% RSLogix 500 project P6.RSS, saved by version 12.00.00.00 %
PROJECT "UNTITLED"    % processor: Bul.1763 MicroLogix 1100 Series B %

PROGRAM FILES
  LAD 2 "MAIN"  3 rungs
  LAD 3 "DIGITAL IO"  2 rungs
  LAD 4 "CONTROL"  10 rungs

DATA FILES
  O0 OUTPUT  4 elements
  I1 INPUT  6 elements
  S2 STATUS  66 elements
  B3 BINARY  1 elements
  T4 TIMER  1 elements
  C5 COUNTER  3 elements
  R6 CONTROL  1 elements
  N7 INTEGER  4 elements
  F8 FLOAT  1 elements

LADDER 2 "MAIN"
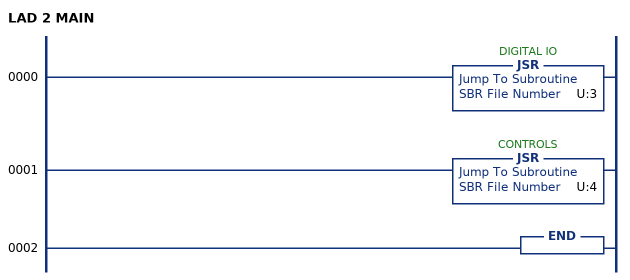
% Rung: 0 %
SOR JSR U:3 EOR
%   U:3  "DIGITAL IO" %
% Rung: 1 %
SOR JSR U:4 EOR
%   U:4  "CONTROLS" %
% Rung: 2 %
SOR END EOR

LADDER 3 "DIGITAL IO"
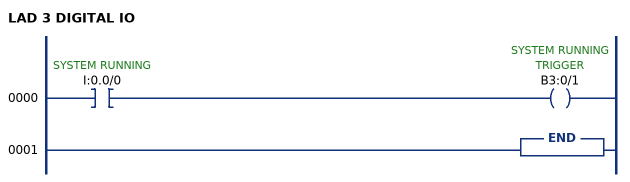
% Rung: 0 %
SOR XIC I:0.0/0 OTE B3:0/1 EOR
%   I:0.0/0  "SYSTEM RUNNING" %
%   B3:0/1  "SYSTEM RUNNING TRIGGER" %
% Rung: 1 %
SOR END EOR

LADDER 4 "CONTROL"
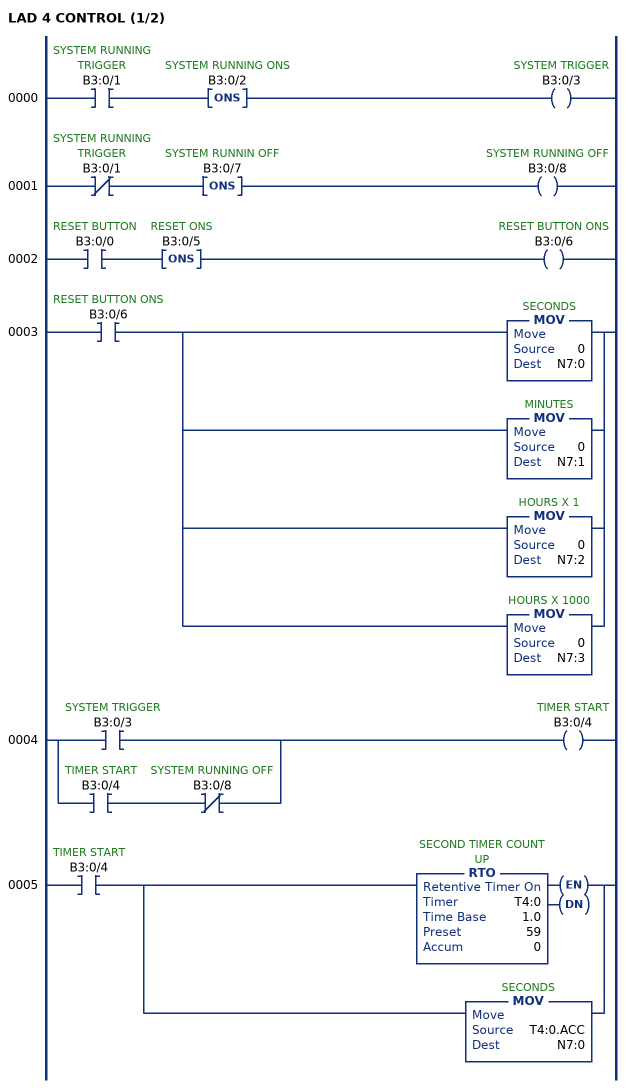
% Rung: 0 %
SOR XIC B3:0/1 ONS B3:0/2 OTE B3:0/3 EOR
%   B3:0/1  "SYSTEM RUNNING TRIGGER" %
%   B3:0/2  "SYSTEM RUNNING ONS" %
%   B3:0/3  "SYSTEM TRIGGER" %
% Rung: 1 %
SOR XIO B3:0/1 ONS B3:0/7 OTE B3:0/8 EOR
%   B3:0/1  "SYSTEM RUNNING TRIGGER" %
%   B3:0/7  "SYSTEM RUNNIN OFF" %
%   B3:0/8  "SYSTEM RUNNING OFF" %
% Rung: 2 %
SOR XIC B3:0/0 ONS B3:0/5 OTE B3:0/6 EOR
%   B3:0/0  "RESET BUTTON" %
%   B3:0/5  "RESET ONS" %
%   B3:0/6  "RESET BUTTON ONS" %
% Rung: 3 %
SOR XIC B3:0/6 BST MOV 0 N7:0 NXB MOV 0 N7:1 NXB MOV 0 N7:2 NXB MOV 0 N7:3 BND EOR
%   B3:0/6  "RESET BUTTON ONS" %
%   N7:0  "SECONDS" %
%   N7:1  "MINUTES" %
%   N7:2  "HOURS X 1" %
%   N7:3  "HOURS X 1000" %
% Rung: 4 %
SOR BST XIC B3:0/3 NXB XIC B3:0/4 XIO B3:0/8 BND OTE B3:0/4 EOR
%   B3:0/3  "SYSTEM TRIGGER" %
%   B3:0/4  "TIMER START" %
%   B3:0/8  "SYSTEM RUNNING OFF" %
% Rung: 5 %
SOR XIC B3:0/4 BST RTO T4:0 1.0 59 0 NXB MOV T4:0.ACC N7:0 BND EOR
%   B3:0/4  "TIMER START" %
%   T4:0  "SECOND TIMER COUNT UP" %
%   N7:0  "SECONDS" %

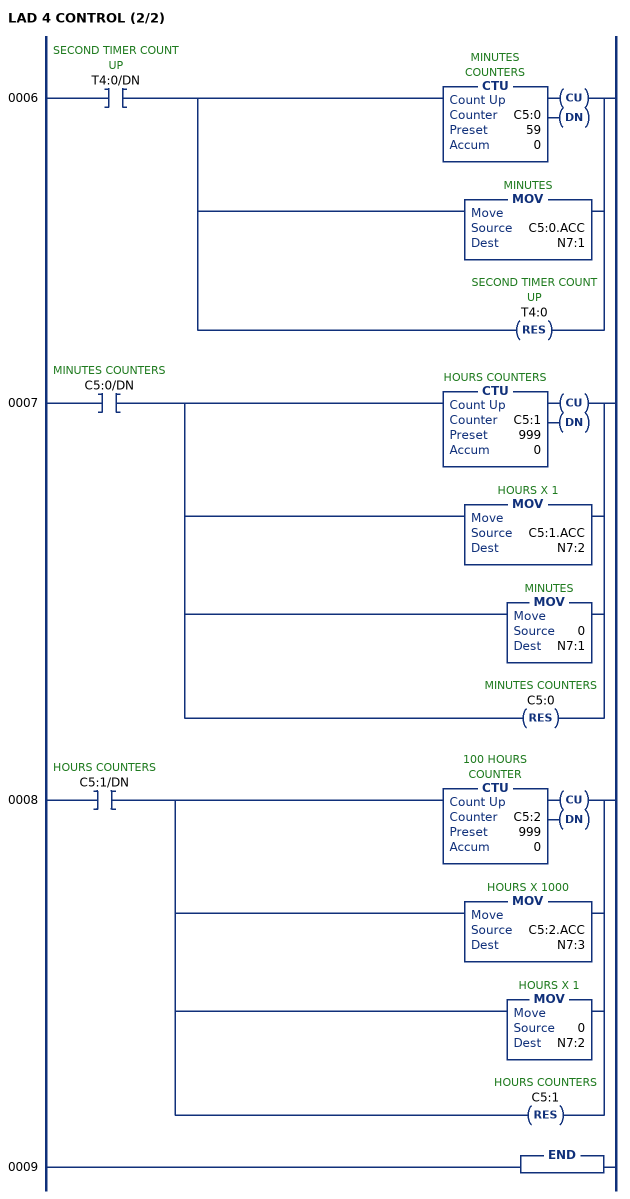
% Rung: 6 %
SOR XIC T4:0/DN BST CTU C5:0 59 0 NXB MOV C5:0.ACC N7:1 NXB RES T4:0 BND EOR
%   T4:0  "SECOND TIMER COUNT UP" %
%   C5:0  "MINUTES COUNTERS" %
%   C5:0.ACC  "SECOND COUNTERS" %
%   N7:1  "MINUTES" %
% Rung: 7 %
SOR XIC C5:0/DN BST CTU C5:1 999 0 NXB MOV C5:1.ACC N7:2 NXB MOV 0 N7:1 NXB RES C5:0 BND EOR
%   C5:0  "MINUTES COUNTERS" %
%   C5:1  "HOURS COUNTERS" %
%   N7:2  "HOURS X 1" %
%   N7:1  "MINUTES" %
% Rung: 8 %
SOR XIC C5:1/DN BST CTU C5:2 999 0 NXB MOV C5:2.ACC N7:3 NXB MOV 0 N7:2 NXB RES C5:1 BND EOR
%   C5:1  "HOURS COUNTERS" %
%   C5:2  "100 HOURS COUNTER" %
%   N7:3  "HOURS X 1000" %
%   N7:2  "HOURS X 1" %
% Rung: 9 %
SOR END EOR

DATA TABLE (non-zero values as saved)
DATA T4
% .PRE .ACC %
% T4:0 % 59 0
DATA C5
% .PRE .ACC %
% C5:0 % 59 0
% C5:1 % 999 0
% C5:2 % 999 0
